PROGRAM SafetyCheck
VAR
	// slave robot information, including arm status and cartesian data
	m_slaveStatus AT %I* :ST_slaveStatus;
	
	// slave robot joint data
	m_slaveJointData AT %I* :ST_slaveJointData;
	
	// setup robot information
	m_setupStatus AT %I* :ST_SetupStatus;
	
	// setup robot joint data
	m_setupJointsData AT %I* :ST_SetupJointData;
	
	//master robot information
	m_masterStatus AT %I* :ST_MasterStatus;
	
	// error check result
	m_safetyCheckData AT %Q* :ST_SafetyData;
	
	// Output cart status
	m_cartStatus AT%I* : ST_CartStatus;
	
	// cart joint data
	m_cartJointsData AT %I* :ST_CartJointData;
	
	//emergency stop and stop botton
	m_stopButton AT %I*: BOOL;
	m_emergencyStopButton AT %I*: BOOL;
	
	//warning tone
	m_warningTone AT %Q*:ARRAY [1..4] OF BOOL;
	
	m_initFlag:bool;
	
	m_SafetyCheck : Fb_SafetyCheck;
	m_checkVariable : ARRAY[1..g_maxNum] OF checkInputVariable;
	m_EtherCATCheck :ARRAY [1..g_maxNum,1..g_maxArmJoint] OF Fb_EtherCATCheck;
	m_errCode :ARRAY [1..3] OF UDINT;
	i , j: INT;
	
	//error robot data record
	m_dataRecord : Fb_dataRecord;
	
	// original position of remote center point when fisrt enter hold state
	m_dsrRcpPos :ARRAY[1..g_sArmNum] OF Vec3d;
	m_rcpPosErrCounts :ARRAY[1..g_sArmNum] OF INT := [4(0)];
	m_rcpPosErr :ARRAY[1..g_sArmNum] OF Vec3d;		// rcp position error
	
	m_armsRS:ARRAY [1..g_maxArmNum,1..30] OF RS;//复位优先双稳态器
	m_cartRS:ARRAY [1..30] OF RS;//复位优先双稳态器
	m_scopeArmNoReady : BOOL;
	
	// wait time before robot init  for ethercat to be statble 
	m_safetyCheckInitWaitTime : LREAL:=0;
END_VAR

// reset data
IF FALSE = m_initFlag  THEN
	FOR i:=1  TO g_sArmNum DO 
		m_safetyCheckData.m_slaveErrFlag[i]:=FALSE;
		m_safetyCheckData.m_setupErrFlag[i]:=FALSE;
		m_safetyCheckData.m_cartErrFlag:=FALSE;
	END_FOR
	m_initFlag:=TRUE;
END_IF

armSafetyCheckInputCast();

armSafetyCheckAllowed();

robotPromptMassageCast();

// wait communication to be stable
IF(m_safetyCheckInitWaitTime<g_robotSafetyCheckWaitTime) THEN
	m_safetyCheckInitWaitTime := m_safetyCheckInitWaitTime+g_setupArmCtrlCycleTime;
	RETURN;
END_IF


FOR i:=1  TO g_maxNum DO
	m_SafetyCheck.systemSafetyCheck(i,m_checkVariable,m_cartJointsData,m_setupJointsData,m_slaveJointData);
END_FOR


//error flag to control
readErrFlag();

//Fault code for UI
m_SafetyCheck.errCodeUpdating();

//The fault code is sent to the UI
GVL_interactUI.g_errIdType3:=m_SafetyCheck.o_ErrCode[3];
GVL_interactUI.g_errIdType2:=m_SafetyCheck.o_ErrCode[2];
GVL_interactUI.g_errIdType1:=m_SafetyCheck.o_ErrCode[1];

//clear fault
IF GVL_interactUI.g_uiFaultReset=1 THEN
	m_SafetyCheck.errFlagReset();
	GVL_interactUI.g_uiFaultReset := 0;
END_IF

//robot record information
//m_dataRecord.run(m_checkVariable , m_cartStatus , m_cartJointsData , m_setupStatus , m_slaveStatus , m_setupJointsData , m_slaveJointData );

m_warningTone := warningTone();

METHOD armSafetyCheckAllowed : BOOL
VAR_INPUT
END_VAR
VAR
	i , j : INT; 
END_VAR

FOR i := 1 TO g_maxArmNum DO
	FOR j := 1 TO g_maxArmJoint DO
		IF j > 5 THEN
			//fault code 16#3003 
			m_SafetyCheck.checkPermit[i].m_linkEncErr[j] := m_checkVariable[i].m_slaveDriverInput[j-g_setupJntNum].m_statusWord<>0;
			//fault code 16#3002 
			m_SafetyCheck.checkPermit[i].m_currentIsNotUpdate[j] :=m_checkVariable[i].m_slaveDriverInput[j-g_setupJntNum].m_statusWord<>0 AND j > 2;
			//fault code 16#2002
			m_SafetyCheck.checkPermit[i].m_armJntFollowErr[j] := m_checkVariable[i].m_slaveDriverInput[j-g_setupJntNum].m_statusWord = DriverStatusWord_OP AND j > 2;
		ELSE
			//fault code 16#3003 
			m_SafetyCheck.checkPermit[i].m_linkEncErr[j] := m_checkVariable[i].m_setupDriverInput[j].m_statusWord<>0;
			//fault code 16#3002
			m_SafetyCheck.checkPermit[i].m_currentIsNotUpdate[j] := m_checkVariable[i].m_setupDriverInput[j].m_statusWord<>0 AND j > 2;
			//fault code 16#2002
			m_SafetyCheck.checkPermit[i].m_armJntFollowErr[j] := m_checkVariable[i].m_setupDriverInput[j].m_statusWord = DriverStatusWord_OP AND j > 2;
			
		END_IF
		//fault code 16#3002
		m_SafetyCheck.checkPermit[i].m_jntStatusErr[j] := TRUE;
		//fault code 16#3004
		m_SafetyCheck.checkPermit[i].m_driveErr[j] := TRUE;
		//fault code 16#3005
		m_SafetyCheck.checkPermit[i].m_armJntEncErr[j] := TRUE;
		//fault code 16#2003
		m_SafetyCheck.checkPermit[i].m_jntVelErr[j] := TRUE;
		//fault code 16#2004
		m_SafetyCheck.checkPermit[i].m_spacePoseErr[j] := m_slaveStatus.m_armState[i] = SlaveArmState_MasterSlave AND  norm(m_slaveStatus.m_masterSlavePoseError[i])<g_smallNum;
		//fault code 16#2005
		m_SafetyCheck.checkPermit[i].m_jntCurrentErr[j] := TRUE;
		//fault code 16#2007
		m_SafetyCheck.checkPermit[i].m_fixedPointErr := m_slaveStatus.m_armState[i] = SlaveArmState_MasterSlave;
		//fault code 16#2008
		m_SafetyCheck.checkPermit[i].m_cmdJntSaltation[j] := m_slaveStatus.m_armState[i] = SlaveArmState_MasterSlave;
		//fault code 16#200C
		m_SafetyCheck.checkPermit[i].m_jntCurrentCtrlErr[j] := m_checkVariable[i].m_setupDriverOutput[j].m_opMode = DriverOPMode_Trq;
		//fault code 16#200F
		m_SafetyCheck.checkPermit[i].m_instruOpenAngle := FALSE;
	END_FOR
END_FOR
END_METHOD

METHOD armSafetyCheckInputCast : BOOL
VAR_INPUT
END_VAR

VAR
	i , j: INT; 
END_VAR

FOR i := 1 TO g_maxArmNum DO
	//emergency stop 、stop button and ui stop 
	m_checkVariable[i].EmergencyStop := m_emergencyStopButton;
	m_checkVariable[i].PCStopButton := GVL_interactUI.g_stopButtonFormUI;
	m_checkVariable[i].SlaveStopButton := m_stopButton;
	//m_SafetyCheck.AlarmVar[i].MasterStopButton
	
	IF m_setupStatus.m_armState[i] <> SetupArmState_Hold THEN
		m_dsrRcpPos[i] := m_setupStatus.m_rcPos[i];
	END_IF
	
	m_checkVariable[i].m_rcpCheck := m_SafetyCheck.rcpErrCheck(m_dsrRcpPos[i],  m_setupStatus.m_rcPos[i], m_rcpPosErrCounts[i] ,m_rcpPosErr[i]);
	m_checkVariable[i].m_spacePoseErr := m_SafetyCheck.poseErrCheck(m_slaveStatus.m_cmdArmPose[i], m_slaveStatus.m_simArmPose[i] );
	
	FOR j:=1 TO  g_sJntNum DO 		
		m_checkVariable[i].m_slaveDriverInput[j] := SlaveArmControl.m_slaveRobot.m_slaveArms[i].m_joints[j].m_motorInputs;
		//3 joint drive error word at number 6 , move one bit to the right to align with the other joints
		IF j = 3 THEN
			m_checkVariable[i].m_slaveDriverInput[j].m_driverError := SHR(SlaveArmControl.m_slaveRobot.m_slaveArms[i].m_joints[j].m_motorInputs.m_driverError,1);
		END_IF
		m_checkVariable[i].m_slaveDriverOutput[j] := SlaveArmControl.m_slaveRobot.m_slaveArms[i].m_joints[j].m_motorOutputs;
		m_checkVariable[i].m_EtherCATState[j+g_setupJntNum] := m_EtherCATCheck[i,j+g_setupJntNum].EtherCATVerify(g_ArmNetID[i],g_JointNetPort[j+g_setupJntNum]);
	END_FOR
	
	FOR j:=1 TO  g_setupJntNum DO 		
		m_checkVariable[i].m_setupDriverInput[j] := SetupArmControl.m_setupRobot.m_setupArms[i].m_joints[j].m_motorInputs;
		m_checkVariable[i].m_setupDriverOutput[j] := SetupArmControl.m_setupRobot.m_setupArms[i].m_joints[j].m_motorOutputs;
		m_checkVariable[i].m_EtherCATState[j] := m_EtherCATCheck[i,j].EtherCATVerify(g_ArmNetID[i],g_JointNetPort[j]);
	END_FOR

END_FOR

FOR j:=1 TO  g_cartJntNum DO
	m_checkVariable[5].EmergencyStop := m_emergencyStopButton;
	m_checkVariable[5].PCStopButton := GVL_interactUI.g_stopButtonFormUI;
	m_checkVariable[5].SlaveStopButton := m_stopButton;
	m_checkVariable[5].m_cartDriverInput[j] := CartControl.m_cartRobot.m_slaveCart.m_cartJoints[j].m_motorInputs;
	m_checkVariable[5].m_cartDriverOutput[j] := CartControl.m_cartRobot.m_slaveCart.m_cartJoints[j].m_motorOutputs;
	m_checkVariable[5].m_cartEtherCATState[j] := m_EtherCATCheck[5,j].EtherCATVerify(g_cartNetID,g_cartJointNetPort[j]);
END_FOR
END_METHOD

METHOD joystickAdjust : BOOL
VAR_IN_OUT CONSTANT
	i_joystickValue : vec8d;
END_VAR

VAR
	i : INT;
END_VAR

FOR i := 1 TO 4 DO
	IF i_joystickValue[i] <> 512 THEN
		joystickAdjust := TRUE;
		EXIT;
	END_IF
END_FOR
END_METHOD

METHOD readErrFlag : BOOL
VAR_INPUT
END_VAR

FOR i:=1  TO g_sArmNum DO
	m_safetyCheckData.m_slaveErrFlag[i] := m_SafetyCheck.m_armErrFlag[i,2] OR m_SafetyCheck.m_armErrFlag[i,3];
	m_safetyCheckData.m_setupErrFlag[i] := m_SafetyCheck.m_armErrFlag[i,2] OR m_SafetyCheck.m_armErrFlag[i,3];
END_FOR


m_safetyCheckData.m_cartErrFlag := m_SafetyCheck.m_armErrFlag[g_cartNum,2] OR m_SafetyCheck.m_armErrFlag[g_cartNum,3];
//cart stead foot error flag
m_safetyCheckData.m_cartSteadyFootErr := m_SafetyCheck.m_jntErrFlag[g_cartNum,1,2] OR m_SafetyCheck.m_jntErrFlag[g_cartNum,1,3] 
																	OR m_SafetyCheck.m_jntErrFlag[g_cartNum,2,2] OR m_SafetyCheck.m_jntErrFlag[g_cartNum,2,3] OR m_SafetyCheck.m_jntErrFlag[g_cartNum,0,2];
//cart wheel error flag
m_safetyCheckData.m_cartWheelErr := m_SafetyCheck.m_jntErrFlag[g_cartNum,3,2] OR m_SafetyCheck.m_jntErrFlag[g_cartNum,3,3]
																OR m_SafetyCheck.m_jntErrFlag[g_cartNum,4,2] OR m_SafetyCheck.m_jntErrFlag[g_cartNum,4,3] OR m_SafetyCheck.m_jntErrFlag[g_cartNum,0,2];
//cart stand column error flag
m_safetyCheckData.m_cartStandColumnErr := m_SafetyCheck.m_jntErrFlag[g_cartNum,5,2] OR m_SafetyCheck.m_jntErrFlag[g_cartNum,5,3] OR m_SafetyCheck.m_jntErrFlag[g_cartNum,0,2];
//cart adjust joint contains 6, 7, and 8 joints
m_safetyCheckData.m_cartAdjustErr := m_SafetyCheck.m_jntErrFlag[g_cartNum,6,2] OR m_SafetyCheck.m_jntErrFlag[g_cartNum,6,3] 
															OR m_SafetyCheck.m_jntErrFlag[g_cartNum,7,2] OR m_SafetyCheck.m_jntErrFlag[g_cartNum,7,3]
															OR m_SafetyCheck.m_jntErrFlag[g_cartNum,8,2] OR m_SafetyCheck.m_jntErrFlag[g_cartNum,8,3] OR m_SafetyCheck.m_jntErrFlag[g_cartNum,0,2];
//cart overhang error flag
m_safetyCheckData.m_cartOverhangErr := m_SafetyCheck.m_jntErrFlag[g_cartNum,8,2] OR m_SafetyCheck.m_jntErrFlag[g_cartNum,8,3] OR m_SafetyCheck.m_jntErrFlag[g_cartNum,0,2];
END_METHOD

METHOD robotPromptMassageCast : BOOL
VAR_IN_OUT CONSTANT
END_VAR

VAR
	i : UDINT;
	m_uiCtrlAdjustFlag : BOOL;
	m_uiCtrlJoystickEnable : BOOL;
	m_joysticksTrigger : BOOL;
	instrument: INT;
END_VAR

FOR i := 1 TO 4 DO
	//0*1021
	m_armsRS[i,1](SET:= m_slaveStatus.m_panelClampErrId[i]=1, 
							RESET1:= NOT m_slaveStatus.m_panelInstallStatus[i], 
							Q1=> m_checkVariable[i].m_promptStatus[1]);
	m_checkVariable[i].m_promptLocation[1] := i + 3;
							
	//0*1022		
	m_armsRS[i,2](SET:= m_slaveStatus.m_panelClampErrId[i]=2, 
							RESET1:= NOT m_slaveStatus.m_panelInstallStatus[i], 
							Q1=> m_checkVariable[i].m_promptStatus[2]);
	m_checkVariable[i].m_promptLocation[2] := i + 3;
	
	//0*102D			//0*1023				
	m_armsRS[i,3](SET:= m_slaveStatus.m_instruReadErrId[i]=1, 
							RESET1:= NOT m_slaveStatus.m_instruInstallStatus[i], 
							Q1=> m_checkVariable[i].m_promptStatus[3]);
	m_checkVariable[i].m_promptLocation[3] := i + 3;
						
	//0*1023			//0*1024	
	m_armsRS[i,4](SET:= m_slaveStatus.m_instruReadErrId[i]=2, 
							RESET1:= NOT m_slaveStatus.m_instruInstallStatus[i], 
							Q1=> m_checkVariable[i].m_promptStatus[4]);
	m_checkVariable[i].m_promptLocation[4] := i + 3;
	
	//0*1030  	//0*1025
	m_armsRS[i,5](SET:= m_slaveStatus.m_instruClampErrId[i]=1, 
							RESET1:= NOT m_slaveStatus.m_instruInstallStatus[i], 
							Q1=> m_checkVariable[i].m_promptStatus[5]);
	m_checkVariable[i].m_promptLocation[5] := i + 3;
	
	//0*1031    //0*1026
	m_armsRS[i,6](SET:= m_slaveStatus.m_instruClampErrId[i]=2, 
							RESET1:= NOT m_slaveStatus.m_instruInstallStatus[i], 
							Q1=> m_checkVariable[i].m_promptStatus[6]);
	m_checkVariable[i].m_promptLocation[6] := i + 3;
	
	//0*1028    //0*1027
	m_armsRS[i,7](SET:= m_slaveStatus.m_instruReadErrId[i]=3, 
							RESET1:= NOT m_slaveStatus.m_instruInstallStatus[i], 
							Q1=> m_checkVariable[i].m_promptStatus[7]);
	m_checkVariable[i].m_promptLocation[7] := i + 3;
	
	//0*1024    //0*1028	
	m_armsRS[i,8](SET:=NOT m_slaveStatus.m_selfCheckPass[i] AND m_slaveStatus.m_panelInstallStatus[i], 
							RESET1:= NOT m_armsRS[i,8].SET, 
							Q1=> m_checkVariable[i].m_promptStatus[8]);
	m_checkVariable[i].m_promptLocation[8] := i + 3;
				
	//0*1033   //0*1029
	
	//0*1032   //0*102A
	m_armsRS[i,10](SET:= m_slaveStatus.m_instruInstallStatus[i] AND NOT m_slaveStatus.m_trocarOnFlag[i], 
							RESET1:= NOT m_armsRS[i,10].SET, 
							Q1=> m_checkVariable[i].m_promptStatus[10]);
	m_checkVariable[i].m_promptLocation[10] := i + 3;	
	
	//0*1025   //0*102B
	FOR j:=1 TO g_mArmNum DO 
		IF i = m_masterStatus.m_teleSlaveArmIdx[j] THEN
			m_armsRS[i,11](SET:=m_slaveStatus.m_armState[i] = SlaveArmState_Disable AND m_masterStatus.m_tryMSControl[j] =1, 
									RESET1:= NOT m_armsRS[i,11].SET, 
									Q1=> m_checkVariable[i].m_promptStatus[11]);
			m_checkVariable[i].m_promptLocation[11] := i + 3;
		END_IF
	END_FOR
	
	//0*1026   //0*102C
	FOR j:=1 TO g_mArmNum DO 
		IF i = m_masterStatus.m_teleSlaveArmIdx[j] THEN
			m_armsRS[i,12](SET:=NOT (SlaveArmState_InstruReady<= m_slaveStatus.m_armState[i] OR m_slaveStatus.m_armState[i] <= SlaveArmState_EndoScope) AND m_masterStatus.m_tryMSControl[j] =1, 
									RESET1:= NOT m_armsRS[i,12].SET, 
									Q1=> m_checkVariable[i].m_promptStatus[12]);
			m_checkVariable[i].m_promptLocation[12] := i + 3;
		END_IF
	END_FOR
	
				
	//0*102F   //0*102D
	m_armsRS[i,13](SET:= norm(m_slaveStatus.m_masterSlavePoseError[i]) > g_smallNum AND m_slaveStatus.m_armState[i] = SlaveArmState_MasterSlave, 
							RESET1:= NOT m_armsRS[i,13].SET, 
							Q1=> m_checkVariable[i].m_promptStatus[13]);
	m_checkVariable[i].m_promptLocation[13] := i + 3;
	
	
	//0*1034   //0*102E
	m_armsRS[i,14](SET:= NOT m_cartStatus.m_asepticDeployCompletedFlag AND (m_masterStatus.m_tryMSControl[1] =1 OR m_masterStatus.m_tryMSControl[2] =1),
							RESET1:= NOT m_armsRS[i,14].SET, 
							Q1=> m_checkVariable[i].m_promptStatus[14]);
	m_checkVariable[i].m_promptLocation[14] := i + 3;		
	
	//0*1035   //0*102F
	IF InstruType_endoscope = m_slaveStatus.m_instruStauts[i].m_type AND m_slaveStatus.m_endoscopeMounted THEN
		m_scopeArmNoReady := m_slaveStatus.m_armState[i] <> SlaveArmState_ScopeReady OR m_slaveStatus.m_armState[i] <> SlaveArmState_EndoScope;
	END_IF
	m_armsRS[i,15](SET:= (NOT m_slaveStatus.m_endoscopeMounted OR m_scopeArmNoReady) AND (m_masterStatus.m_tryMSControl[1] =1 OR m_masterStatus.m_tryMSControl[2] =1), 
							RESET1:= NOT m_armsRS[i,15].SET, 
							Q1=> m_checkVariable[i].m_promptStatus[15]);
	m_checkVariable[i].m_promptLocation[15] := i + 3;	
	
END_FOR

//0*102E		 //0*1030			
m_cartRS[16](SET:= NOT m_slaveStatus.m_masterOnLine, 
						RESET1:= m_slaveStatus.m_masterOnLine, 
						Q1=> m_checkVariable[g_cartNum].m_promptStatus[16]);
m_checkVariable[g_cartNum].m_promptLocation[16] := 16#0C;

//0*1027   //0*1031
m_cartRS[17](SET:=m_cartStatus.m_cartDumpEnergy <= 30 , 
						RESET1:= m_cartStatus.m_cartDumpEnergy>30, 
						Q1=> m_checkVariable[g_cartNum].m_promptStatus[17]);
m_checkVariable[g_cartNum].m_promptLocation[17] := g_cartNum + 3;

//0*1029   //0*1032	

//0*102A   //0*1033
m_cartRS[19](SET:= m_cartStatus.m_sdrivingLeverSensorManualFlag, 
						RESET1:=NOT m_cartStatus.m_sdrivingLeverSensorManualFlag, 
						Q1=> m_checkVariable[g_cartNum].m_promptStatus[19]);
m_checkVariable[g_cartNum].m_promptLocation[19] := g_cartNum + 3;

//0*102C   //0*1034
m_uiCtrlJoystickEnable := m_cartStatus.m_uiControl.m_cameraJoystickEnable OR m_cartStatus.m_uiControl.m_joystickEnable;
m_joysticksTrigger := joystickAdjust(m_cartStatus.m_joystickValue);
m_cartRS[20](SET:= m_cartStatus.m_trocarOnFlag=0 AND NOT m_uiCtrlJoystickEnable AND m_joysticksTrigger, 
						RESET1:= NOT m_cartRS[20].SET, 
						Q1=> m_checkVariable[g_cartNum].m_promptStatus[20]);
m_checkVariable[g_cartNum].m_promptLocation[20] := g_cartNum + 3;
					
//0*102B   //0*1035
m_uiCtrlAdjustFlag := m_cartStatus.m_uiControl.m_cameraJoystickEnable OR m_cartStatus.m_uiControl.m_dockingEnable OR m_cartStatus.m_uiControl.m_drapingEnable
							OR m_cartStatus.m_uiControl.m_joystickEnable OR m_cartStatus.m_uiControl.m_packageEnable;
m_cartRS[21](SET:= m_cartStatus.m_trocarOnFlag>0 AND m_uiCtrlAdjustFlag, 
						RESET1:= m_cartStatus.m_trocarOnFlag=0 OR NOT m_uiCtrlAdjustFlag, 
						Q1=> m_checkVariable[g_cartNum].m_promptStatus[21]);
m_checkVariable[g_cartNum].m_promptLocation[21] := g_cartNum + 3;

//0*1036
m_cartRS[22](SET:= m_cartStatus.m_jntPosReachLimit[5] OR m_cartStatus.m_jntPosReachLimit[6] OR m_cartStatus.m_jntPosReachLimit[7] OR m_cartStatus.m_jntPosReachLimit[8], 
						RESET1:= NOT m_cartRS[22].SET, 
						Q1=> m_checkVariable[g_cartNum].m_promptStatus[22]);
m_checkVariable[g_cartNum].m_promptLocation[22] := g_cartNum + 3;
END_METHOD

METHOD warningTone : vec4b
VAR_INPUT
END_VAR

IF (GVL_interactUI.g_curErrType=3) THEN
	warningTone[1] := TRUE;
	warningTone[2] := FALSE;
	warningTone[3] := FALSE;
ELSIF (GVL_interactUI.g_curErrType=2) THEN
	warningTone[1] := FALSE;
	warningTone[2] := TRUE;
	warningTone[3] := FALSE;
ELSIF  (GVL_interactUI.g_curErrType=1) THEN
	warningTone[1] := FALSE;
	warningTone[2] := FALSE;
	warningTone[3] := TRUE;
ELSE
	warningTone[1] := FALSE;
	warningTone[2] := FALSE;
	warningTone[3] := FALSE;
END_IF
END_METHOD

END_PROGRAM

(* stored: Version 1.1.0.1, ProductVersion 3.1.4024.11
   POU SafetyCheck: Id {54e6e883-3f22-4a40-9066-2b433bf8009c}, SpecialFunc None
   Method armSafetyCheckAllowed: Id {c2ebef6f-e712-49e3-9955-377a0083e93a}
   Method armSafetyCheckInputCast: Id {598e934b-b439-4bef-985d-1ea697c2fcb0}
   Method joystickAdjust: Id {38ce96d9-75fc-4e3b-9d39-89b30533a7ac}
   Method readErrFlag: Id {c6c3fbb5-bc5f-41ea-91b5-687651d637ca}
   Method robotPromptMassageCast: Id {4528e69f-5454-4a94-84aa-1a99d7ab54e4}
   Method warningTone: Id {82112973-2b93-4990-831a-9a609be275a4} *)
